FUNCTION_BLOCK TOnTimer
VAR
    TON1 : TON;
END_VAR

METHOD Delay : BOOL
VAR_INPUT
    In : BOOL;
END_VAR
TON1(IN := In);
Delay := TON1.Q;
END_METHOD

METHOD FB_init : BOOL
VAR_INPUT
	bInitRetains : BOOL; // if TRUE, the retain variables are initialized (warm start / cold start)
	bInCopyCode : BOOL;  // if TRUE, the instance afterwards gets moved into the copy code (online change)
    PresetTime : LREAL; // seconds
END_VAR
TON1.PT := LREAL_TO_TIME(PresetTime * 1000);
END_METHOD

PROPERTY OutputState : BOOL
GET
OutputState := TON1.Q;
END_GET
END_PROPERTY

PROPERTY PresetTime : LREAL
GET
PresetTime := TIME_TO_LREAL(TON1.PT)/1000.0; // in seconds
END_GET
SET
TON1.PT := LREAL_TO_TIME(PresetTime * 1000);
END_SET
END_PROPERTY

METHOD Reset
TON1(IN := FALSE);
END_METHOD

METHOD Run : BOOL
TON1(IN := TRUE);
Run := TON1.Q;
END_METHOD

END_FUNCTION_BLOCK

(* stored: Version 1.1.0.1, ProductVersion 3.1.4024.3
   POU TOnTimer: Id {124c9a8e-014d-0bbe-2276-3abf7760eeb2}, SpecialFunc None
   Method Delay: Id {78a602f0-5cc4-0d95-13a2-8f01cd3d694c}
   Method FB_init: Id {270a6cd2-c16c-0b13-1a36-751302649b14}
   Property OutputState: Id {d7b83ff1-258e-4688-84b0-85322bc7596d}
   Get Get: Id {c2125d2f-97e5-4d16-8d04-1044ed147f9a}
   Property PresetTime: Id {b0441a1c-a168-0c1b-2899-7925e3bff834}
   Get Get: Id {76eae6fc-dfdf-0bfd-1e48-baacbed5e95f}
   Set Set: Id {dbfa754f-7d5f-0c31-1944-e57c0c36cfe7}
   Method Reset: Id {bf1ce0ca-ddda-0a0e-2ec5-8f64ee894393}
   Method Run: Id {015a040d-e1c7-0001-3207-3310fc552742} *)
